# B&R Automation Studio project webdemo
Automation Studio 4.5.2.102

## Configuration Simulation

CPU X20CP3585, AutomationRuntime V4.08, Build 4.1.2, Safety 0.0

### Task classes (Cpu.sw)
```
Cyclic#4:
  webdata <- WebServer.webdata.prg
Binaries: iomap, sysconf, arconfig, ashwd, asfw
Libraries: Runtime
```

### Hardware
```
X20BM11 : X20BM11 v1.0.0.1  [X2X1 -> X20CP3585.IF6]
X20CP3585 : X20CP3585 v1.3.0.0
  Connector IF2:
    ActivateDevice = 1
    EthInterfaceRedundant = 0
    HostName = if2-mycp3585
    Mode = Manual
    InternetAddress = 10.49.40.221
    SubnetMask = 255.255.255.0
  Connector IF3:
    EplInterfaceRedundant = 0
    EplHostName = if3-mycp3585
    EplEthInterfaceRedundant = 0
    HostName = if3-eth-mycp3585
  Connector IF6:
    CycleTime = 10000
  ConfigurationID = webdemo_X20CP
  Simulation = 1
  EnableUsbRemoteInstall = 1
  EthernetHostName = mycp3585
  FtpUser1
  FtpUsername1 = ich
  FtpUserPassword1 = PsbtO9eSDR2PTXLzf1bU4yBAucIjxDv5zVoWpEx6m9g=
  FtpUserSalt1 = 1FNSeuv6
  FTPAccessRight1 = 0
  FTPdevice1 = ALL
  WebServerWebDir = C:\Users\hilchenbachc\Documents\asprojekte\drehmo\webdemo\CompactFlash\web
  SdmColor = colorRGB
  SdmColorR = 0
  SdmColorG = 129
  SdmColorB = 227
X20DO9321 : X20DO9321 v1.0.2.0  [SS1 -> X20TB12.SS; SL -> X20BM11.SL1]
  Supervision = off
X20TB12 : X20TB12 v1.0.0.0
```

### IoMap.iom - X20CP3585/IoMap.iom
```iecst
(********************************************************************
 * COPYRIGHT -- Bernecker + Rainer
 ********************************************************************
 * Datei: IoMap.iom
 * Autor: hilchenbachc
 * Erstellt: 18. Februar 2015
 ********************************************************************
 * IO-Rangierungsdatei
 ********************************************************************)
VAR_CONFIG
	WebPV.btnPlus AT %QX."X20DO9321".DigitalOutput03;
	WebPV.btnMinus AT %QX."X20DO9321".DigitalOutput04;
	::WebPV.bool1 AT %QX."X20DO9321".DigitalOutput01;
	::WebPV.bool2 AT %QX."X20DO9321".DigitalOutput02;
END_VAR
```

## Configuration X20CP

CPU X20CP3585, AutomationRuntime D4.52, Build 4.1.2, Safety 0.0

### Hardware
```
X20BM11 : X20BM11 v1.0.0.1  [X2X1 -> X20CP3585.IF6]
X20CP3585 : X20CP3585 v1.3.0.0
  Connector IF2:
    ActivateDevice = 1
    Mode = Manual
    InternetAddress = 192.168.0.10
    SubnetMask = 255.255.255.0
  Connector IF3:
    EplHostName = br-automation
    HostName = br-automation
  Connector IF6:
    CycleTime = 10000
  ConfigurationID = webdemo_X20CP
  UserPartitionSize = 100
  Simulation = 1
  WebServerWebDir = C:\projects\webdemo\USER\web
  SdmColor = colorRGB
  SdmColorR = 0
  SdmColorG = 129
  SdmColorB = 227
X20DO9321 : X20DO9321 v1.0.2.0  [SS1 -> X20TB12.SS; SL -> X20BM11.SL1]
  Supervision = off
X20TB12 : X20TB12 v1.0.0.0
```

## Logical view

Binary libraries used (declarations not repeated): operator, runtime, astime, AsIecCon


### Package Logical/WebServer - WebServer

### WebServer.typ - Package data types
```iecst
(********************************************************************
 * COPYRIGHT -- Bernecker + Rainer
 ********************************************************************
 * Package: WebServer
 * File: WebServer.typ
 * Author: hilchenbachc
 * Created: February 02, 2015
 ********************************************************************
 * Data types of package WebServer
 ********************************************************************)

TYPE
	WebPVCyclicTyp : 	STRUCT
		currentTime : UDINT;
	END_STRUCT;
	WebPVTyp : 	STRUCT
		cyclic : WebPVCyclicTyp;
		test1 : REAL;
		test2 : REAL;
		bool1 : BOOL;
		bool2 : BOOL;
		range1 : REAL;
		btnPlus : BOOL;
		btnMinus : BOOL;
		array : ARRAY[0..19]OF REAL;
	END_STRUCT;
END_TYPE
```

### WebServer.var - Package variables
```iecst
(********************************************************************
 * COPYRIGHT -- Bernecker + Rainer
 ********************************************************************
 * Package: WebServer
 * File: WebServer.var
 * Author: hilchenbachc
 * Created: February 02, 2015
 ********************************************************************
 * Variables of package WebServer
 ********************************************************************)
VAR
	WebPV : WebPVTyp := (0);
END_VAR
```

### Program Logical/WebServer/webdata (IEC) - Daten fuer den Webserver

#### webdata.st - Implementierungscode
```iecst
(********************************************************************
 * COPYRIGHT -- Bernecker + Rainer
 ********************************************************************
 * Programm: webdata
 * Datei: webdata.st
 * Autor: hilchenbachc
 * Erstellt: 30. Januar 2015
 ********************************************************************
 * Implementierung des Programms webdata
 ********************************************************************)

PROGRAM _INIT

	DTGetTime_1.enable:=1;
	WebPV.test1 := 3.14;

END_PROGRAM

PROGRAM _CYCLIC
	(* aktuelle Uhrzeit *)
	DTGetTime_1();
	WebPV.cyclic.currentTime := DT_TO_UDINT(DTGetTime_1.DT1);

	WebPV.test2 := WebPV.test2 + 1.31;
	IF( WebPV.test2 > 100.0 ) THEN
		WebPV.test2 := -100;
	END_IF

	WebPV.array[0] := WebPV.array[0] + 1.422;

	FOR i:= 1 TO 19 DO
		WebPV.array[i] := WebPV.array[0] * i*2.1;
	END_FOR

END_PROGRAM
```

#### webdata.var - Lokale Variablen
```iecst
(********************************************************************
 * COPYRIGHT -- Bernecker + Rainer
 ********************************************************************
 * Programm: webdata
 * Datei: webdata.var
 * Autor: hilchenbachc
 * Erstellt: 30. Januar 2015
 ********************************************************************
 * Lokale Variablen des Programms webdata
 ********************************************************************)
VAR
	DTGetTime_1 : DTGetTime;
	i : INT;
END_VAR
```
